PROGRAM P_Notifications
VAR
END_VAR

END_PROGRAM

(* stored: Version 1.1.0.1
   POU P_Notifications: Id {8e195bf0-9a3a-4b45-b03a-44b3843a5af3}, SpecialFunc None *)
